(* CODESYS project Machine_Expert_ Template.project
   Version: 0.0.0.0
   Title: Machine_Expert_ Template
   Author: HP

Project tree, tasks and I/O mapping:
  MyController : TM241CE24T/U, Schneider Electric, order no. TM241CE24T/U, version 5.0.8.2
    application Application
      task MAST (cyclic, interval 20 ms, priority 15, watchdog 100 ms x 1) calls nothing
      global variables GVL
      program POU_Ladder [LD]
    DI : Digital Inputs, Schneider Electric, version 5.0.8.2
        input  iwDI_IW0 : WORD  // IW0
        input  ibDI_IB1 : BYTE  // IB1
    DQ : Digital Outputs, Schneider Electric, version 5.0.8.2
        output qwDQ_QW0 : WORD  // QW0
        output qbDQ_QB1 : BYTE  // QB1
    Counters : Counters, Schneider Electric, version 5.0.8.2
    Pulse_Generators : Pulse Generators, Schneider Electric, version 5.0.8.2
    Cartridge_1 : Cartridge, Schneider Electric, version 5.0.8.2
    IO_Bus : IO bus - TM3, Schneider Electric, version 5.0.8.2
      Module : TM3DI8/G, Schneider Electric, order no. TM3DI8/G, version 1.0.1.11
          input  ibModule_IB0 : BYTE  // IB0
    COM_Bus : COM bus, Schneider Electric, version 5.0.8.2
    Ethernet_1 : Ethernet Network, Schneider Electric, version 5.0.8.2
    Serial_Line_1 : Serial line, Schneider Electric, version 5.0.8.2
      Machine_Expert_Network_Manager : Machine Expert-Network Manager, Schneider Electric, version 4.0.0.3
    Serial_Line_2 : Serial line, Schneider Electric, version 5.0.8.2
      Modbus_Manager : Modbus Manager, Schneider Electric, version 4.0.0.3
*)

// MyController/Application/GVL
{attribute 'qualified_only'}
VAR_GLOBAL
END_VAR

// MyController/Application/POU_Ladder
PROGRAM POU_Ladder
VAR
	emergency_pb AT %IX0.0: BOOL;
	TON_0: TON;
	System_ready AT %M0: BOOL;
	Input_1 AT %IX0.1: BOOL;
	Output_1 AT %QX0.0: BOOL;
END_VAR

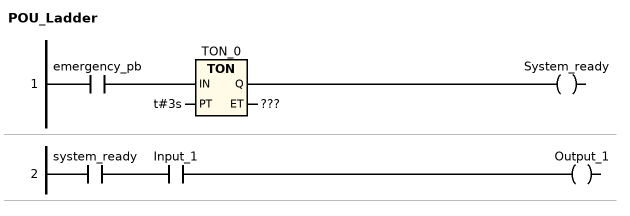
// NETWORK 1
TON_0(IN := emergency_pb, PT := t#3s); // TON
System_ready := TON_0.Q;

// NETWORK 2
Output_1 := system_ready AND Input_1;

END_PROGRAM
